TYPE PathMotionParameters_typ :
STRUCT
	
	Jerk				: LREAL;
	Acceleration		: LREAL;
	Deceleration		: LREAL;
	Velocity			: LREAL;
	
	BlendingRadii		: ARRAY[0..1] OF LREAL;

END_STRUCT
END_TYPE

(* stored: Version 1.1.0.1, ProductVersion 3.1.4024.9
   DUT PathMotionParameters_typ: Id {842b757e-ba1c-4730-8853-8fb8fa7d7d60} *)
